FUNCTION_BLOCK MATRIX
VAR_INPUT
	x1, x2, x3, x4, X5 : BOOL;
END_VAR
VAR_INPUT CONSTANT
	Release : BOOL;
END_VAR
VAR_OUTPUT
	code : BYTE;
	TP : BOOL;
	y1: BOOL := TRUE;
	y2, y3, y4 : BOOL;
END_VAR
VAR
	line : BYTE;
	X : ARRAY[0..3] OF BYTE; (* scan line inputs *)
	L : ARRAY[0..3] OF BYTE; (* scan line status *)
	i: INT;
	temp: BYTE;
END_VAR

(*
version 1.3	26 oct. 2008
programmer 	hugo
tested by	oscat

MATRIX is a matrix keyboard encoder for 4 rows and up to 5 columns.
matrix can send a code while a key is pressed and it sends another code while a key is released when the setup variable 'release' is set to true.
the setup variable release is false the code is only sent when the key is pressed.
the output byte holds the 5 columns in the lowest bits 0..2  and the row number in bits 4..6, while bit 7 is true for a key pressed and false for a key released.

*)

TP := FALSE;
CODE := 0;
(* read scan lines *)
X[line].0 := X1;
X[line].1 := X2;
X[line].2 := X3;
X[line].3 := X4;
X[line].4 := X5;

(* compare for change *)
FOR i := 0 TO 3 DO
	IF X[i] <> L[i] THEN
		(* scan line information has changed code need to be found and generated *)
		temp := x[i] XOR L[i];
		IF temp.0 THEN
			CODE := 1;
			code.7 := X[i].0;
			L[i].0 := X[i].0;
		ELSIF temp.1 THEN
			code := 2;
			code.7 := X[i].1;
			L[i].1 := X[i].1;
		ELSIF temp.2 THEN
			code := 3;
			code.7 := X[i].2;
			L[i].2 := X[i].2;
		ELSIF temp.3 THEN
			CODE := 4;
			CODE.7 := X[i].3;
			L[i].3 := X[i].3;
		ELSIF temp.4 THEN
			CODE := 5;
			CODE.7 := X[i].4;
			L[i].4 := X[i].4;
		END_IF;
		TP := TRUE;
		CODE.4 := Line.0;
		CODE.5 := Line.1;
		CODE.6 := Line.2;

		(* check if release codes need to be killed *)
		IF NOT release AND CODE < 127 THEN
			CODE := 0;
			TP := FALSE;
		END_IF;
		EXIT;
	END_IF;
END_FOR;

(* increment scan line every cycle *)
line := (line + 1) AND 2#0000_0011;
temp := SHL(BYTE#1,line);
Y1 := temp.0;
Y2 := temp.1;
Y3 := temp.2;
Y4 := temp.3;




(* revision history
hm		10.6.2007	rev 1.0		
	original version 


hm		11.9.2007	rev 1.1		
	deleted unused variables k and old_code

hm		23.12.2007	rev 1.2
	added exit statement in for loop instead of i:=5

hm		26. oct. 2008	rev 1.3
	code optimized

*)

END_FUNCTION_BLOCK

(* stored: Version 1.1.0.1, ProductVersion 3.1.4022.7
   POU MATRIX: Id {5f23ab1d-cba1-4180-b243-d4839731a243}, SpecialFunc None *)
